(* PLC project PLC, Beckhoff Automation GmbH TwinCAT PLC Control 3.5.13.21 *)
(* stored: creationDateTime 2024-02-17T22:43:37.076425, modificationDateTime 2024-02-17T22:43:37.076425 *)

PROGRAM MAIN
VAR
	// resources
	cylinders: ARRAY[0..G.numAxis] OF CylResource;
	PBs: ARRAY[0..G.numAxis] OF PBResource;
	LPs: ARRAY[0..G.numAxis] OF LPResource;
	
	// system
	firstScan: BOOL := TRUE;
	
	// 動作設定
	permConfigCyl: ARRAY[0..G.numAxis] OF CylConfig;
	permConfigPB: ARRAY[0..G.numAxis] OF PBConfig;
	permConfigLP: ARRAY[0..G.numAxis] OF LPConfig;
	i: LINT;
	unmatchConfig: BOOL := FALSE;
END_VAR

            Unit();


// 動作設定不一致を調べる
unmatchConfig := FALSE;
FOR i := 0 TO G.numAxis DO
	IF permConfigCyl[i].cylinderErrorTime <> cylinders[i].config.cylinderErrorTime THEN
		unmatchConfig := TRUE;
	END_IF
	IF permConfigCyl[i].operateDelayTime <> cylinders[i].config.operateDelayTime THEN
		unmatchConfig := TRUE;
	END_IF
	IF permConfigCyl[i].sensorDelayTime <> cylinders[i].config.sensorDelayTime THEN
		unmatchConfig := TRUE;
	END_IF
	IF permConfigPB[i].pushDelayTime <> PBs[i].config.pushDelayTime THEN
		unmatchConfig := TRUE;
	END_IF
	IF permConfigLP[i].invert <> LPs[i].config.invert THEN
		unmatchConfig := TRUE;
	END_IF
END_FOR


// 起動後初回に動作設定を元に戻す
IF firstScan THEN
	FOR i := 0 TO G.numAxis DO
		cylinders[i].config := permConfigCyl[i];
		PBs[i].config := permConfigPB[i];
		LPs[i].config := permConfigLP[i];
	END_FOR
END_IF


firstScan := FALSE;
          
END_PROGRAM
